Omron CX-Programmer project NewProject (CX-Programmer 9.73)

# PLC NewPLC1: CP1E N20

## Global symbols (name address type ; comment)
0.01 BOOL  ; PB START
0.02 BOOL  ; PB STOP
100.01 BOOL  ; LAMP
100.05 BOOL  ; LAMP
200.01 BOOL  ; KEEP

## Program NewProgram1 (cyclic task 0)

### Section Section1

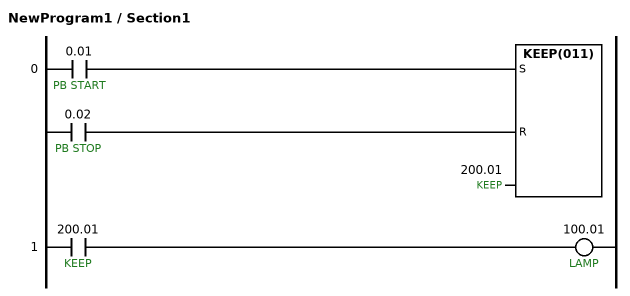
; rung 0
LD 0.01  ; PB START
LD 0.02  ; PB STOP
KEEP(011) 200.01  ; KEEP
; rung 1
LD 200.01  ; KEEP
OUT 100.01  ; LAMP

### Section END
; rung 0
END(001)